SUBAPPLICATION Uebung_231_AX (* 1 Taster via AX_ASR_RF_TRIG + ASR_SPLIT_2 auf 2 unabhaengige ASR_AX_SR-Latches (Q1+Q2) - Spiegelbild zu Uebung_230_AX (dort MERGE N->1, hier SPLIT 1->N) *)
  (* Standard: 61499-2; Description: Copyright (c) 2026 Meisterschulen am Ostbahnhof This program and the accompanying materials are made available under the terms of the Eclipse Public License 2.0 which is available at https://www.eclipse.org/legal/epl-2.0/ SPDX-License-Identifier: EPL-2.0 *)
  (* Version 1.0, 2026-09-07, Franz Höpfinger, Meisterschulen am Ostbahnhof, initial API and implementation and/or initial documentation *)
  PACKAGE Uebungen;
  IMPORT logiBUS::io::DI::logiBUS_DI::Input_I1;
  IMPORT logiBUS::io::DQ::logiBUS_DO::Output_Q1;
  IMPORT logiBUS::io::DQ::logiBUS_DO::Output_Q2;
  (* Documentation:
  1 Taster über ASR_SPLIT_2 auf 2 unabhängige Latches (Fan-out)
   Spiegelbild zu Uebung_230_AX: dort führte ASR_MERGE_2 zwei Quellen zu einem gemeinsamen Latch zusammen (N→1, Fan-in). Hier ist es umgekehrt: ein Taster steuert über ASR_SPLIT_2 zwei unabhängige Latches gleichzeitig (1→N, Fan-out).
   Funktionsbeschreibung
    - AX_ASR_RF_TRIG_1: Taster drücken → SET, loslassen → RESET, als ein einziges gebündeltes ASR-Signal.
   - Warum ASR_SPLIT_2 nötig ist: ein Adapter-Plug (AX_ASR_RF_TRIG_1.Q) ist strikt punkt-zu-punkt - er kann nicht direkt gleichzeitig an zwei ASR_AX_SR.S_R-Sockets angeschlossen werden. Genau dieselbe Grunderegel, die in 229/230 ASR_MERGE_2 nötig machte (mehrere Quellen können nicht direkt auf einen Socket), erzwingt hier umgekehrt ASR_SPLIT_2 (eine Quelle kann nicht direkt zwei Plugs gleichzeitig bedienen).
   - ASR_SPLIT_2 dupliziert den einen ASR-Stream verlustfrei auf ASR_AX_SR_1 und ASR_AX_SR_2 - beide Latches erhalten exakt dieselben SET/RESET-Kommandos zur exakt gleichen Zeit und laufen daher synchron, obwohl sie zwei komplett unabhängige Bausteine mit je eigenem Ausgang (Q1/Q2) sind.
    Arbeitsauftrag
   Testen Sie: Taster I1 drücken und halten → Q1 UND Q2 gleichzeitig EIN. Loslassen → beide gleichzeitig AUS. Beobachten Sie im 4diac-Editor, dass ASR_AX_SR_1 und ASR_AX_SR_2 zwei getrennte Instanzen sind, die nur über den gemeinsamen ASR_SPLIT_2-Ursprung gekoppelt sind - keine direkte Verbindung zwischen ihnen.
  *)
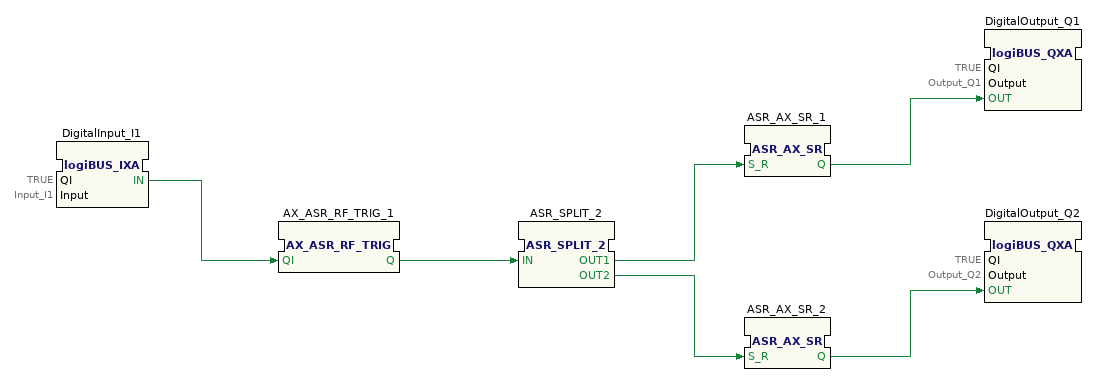
  (* Spiegelbild zu Uebung_230_AX: dort fuehrte ASR_MERGE_2 2 Quellen auf 1 Latch zusammen (N->1), weil ein Adapter-Socket nur eine Quelle annimmt. Hier ist es umgekehrt: AX_ASR_RF_TRIG_1.Q ist auch nur EIN Socket-Ausgang und kann nicht direkt an 2 ASR_AX_SR.S_R gleichzeitig angeschlossen werden - ASR_SPLIT_2 dupliziert den EINEN ASR-Stream auf 2 Ziele (1->N). *)
  FBS
    DigitalInput_I1 : logiBUS::io::DI::logiBUS_IXA(QI := TRUE, Input := Input_I1);
    AX_ASR_RF_TRIG_1 : adapter::events::unidirectional::AX_ASR_RF_TRIG;
    ASR_SPLIT_2 : adapter::events::unidirectional::ASR_SPLIT_2;
    ASR_AX_SR_1 : adapter::events::unidirectional::ASR_AX_SR;
    ASR_AX_SR_2 : adapter::events::unidirectional::ASR_AX_SR;
    DigitalOutput_Q1 : logiBUS::io::DQ::logiBUS_QXA(QI := TRUE, Output := Output_Q1);
    DigitalOutput_Q2 : logiBUS::io::DQ::logiBUS_QXA(QI := TRUE, Output := Output_Q2);
  END_FBS
  ADAPTER_CONNECTIONS
    DigitalInput_I1.IN TO AX_ASR_RF_TRIG_1.QI;
    AX_ASR_RF_TRIG_1.Q TO ASR_SPLIT_2.IN;
    ASR_SPLIT_2.OUT1 TO ASR_AX_SR_1.S_R;
    ASR_SPLIT_2.OUT2 TO ASR_AX_SR_2.S_R;
    ASR_AX_SR_1.Q TO DigitalOutput_Q1.OUT;
    ASR_AX_SR_2.Q TO DigitalOutput_Q2.OUT;
  END_CONNECTIONS
END_SUBAPPLICATION
